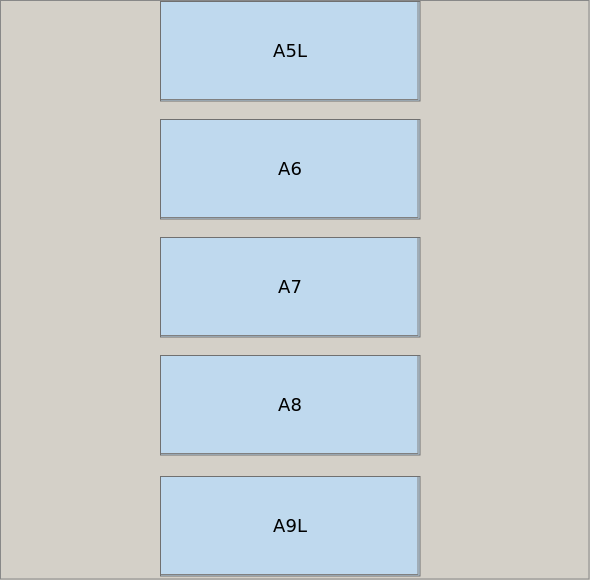
VISUALIZATION tempEflexScreen  // 590x580
    Button (160,1 260x100), "A5L"
        OnMouseDown: execute { tempEflex.nEflexState := 1; }
    Button (160,119 260x100), "A6"
        OnMouseDown: execute { tempEflex.nEflexState := 2; }
    Button (160,237 260x100), "A7"
        OnMouseDown: execute { tempEflex.nEflexState := 3; }
    Button (160,476 260x100), "A9L"
        OnMouseDown: execute { tempEflex.nEflexState := 5; }
    Button (160,355 260x100), "A8"
        OnMouseDown: execute { tempEflex.nEflexState := 4; }
END_VISUALIZATION

(* stored: Version 1.1.0.1, ProductVersion 3.1.4024.15
   Visu tempEflexScreen: Id {89b81827-5f54-4f78-a155-2dba79c74e5b} *)
